// Mitsubishi GX Works2 project: STW_4Counter_Structure_V3   PLC: FX3U/FX3UC

// task Task_01 (event TRUE, interval 0, priority 31): POU_01

PROGRAM POU_01
VAR
  FDCounter_1 : FDCounter;
  FDCounter_2 : FDCounter;
  FDCounter_3 : FDCounter;
  FDCounter_4 : FDCounter;
  FDCounter_5 : FDCounter;
  FDCounter_6 : FDCounter;
  FDCounter_7 : FDCounter;
  FDCounter_8 : FDCounter;
END_VAR
(* structured ladder/FBD written out as ST: instructions are called as NAME(EN, inputs, outputs); _pN, _eN, _tN stand for wires *)
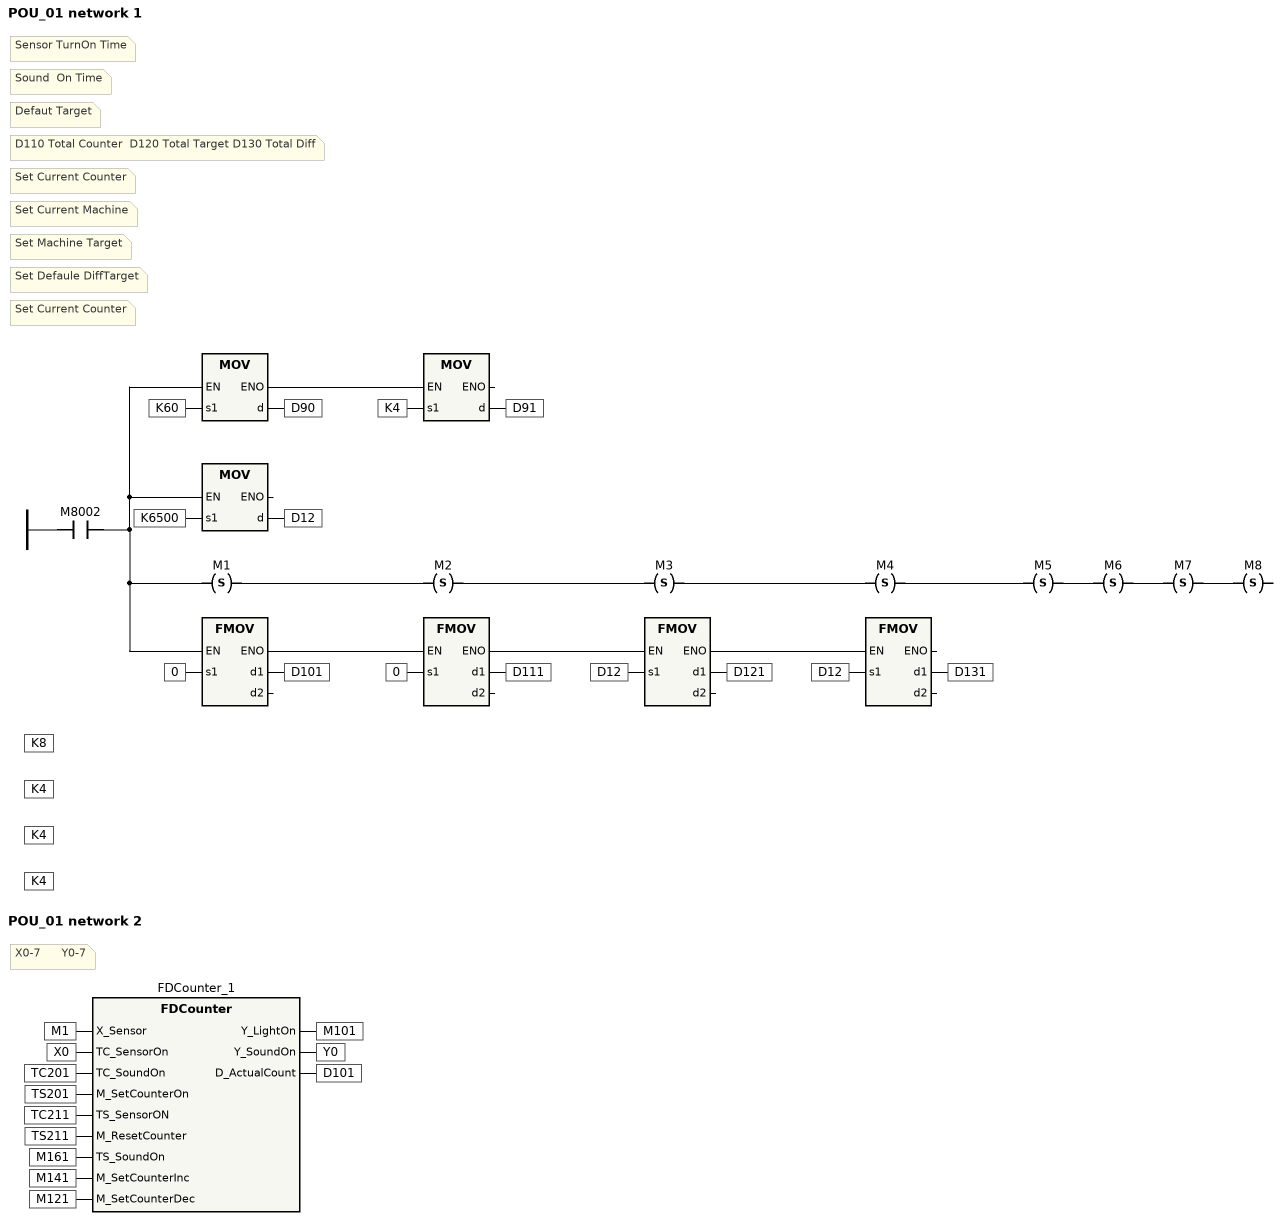
(* network 1 *)
(* Sensor TurnOn Time *)
(* Sound  On Time *)
(* Defaut Target *)
(* D110 Total Counter  D120 Total Target D130 Total Diff *)
(* Set Current Counter *)
(* Set Current Machine *)
(* Set Machine Target *)
(* Set Defaule DiffTarget *)
(* Set Current Counter *)
_e1 := MOV(M8002, K60, D90);
MOV(_e1, K4, D91);
MOV(M8002, K6500, D12);
_e2 := FMOV(M8002, 0, D101, _open);
_e3 := FMOV(_e2, 0, D111, _open);
_e4 := FMOV(_e3, D12, D121, _open);
FMOV(_e4, D12, D131, _open);
SET(M8002, M1);
SET(M8002, M2);
SET(M8002, M3);
SET(M8002, M4);
SET(M8002, M5);
SET(M8002, M6);
SET(M8002, M7);
SET(M8002, M8);
(* not connected to any output: K8, K4, K4, K4 *)
(* network 2 *)
(* X0-7      Y0-7 *)
FDCounter_1(X_Sensor := M1, TC_SensorOn := X0, TC_SoundOn := TC201, M_SetCounterOn := TS201, TS_SensorON := TC211, M_ResetCounter := TS211, TS_SoundOn := M161, M_SetCounterInc := M141, M_SetCounterDec := M121, Y_LightOn => M101, Y_SoundOn => Y0, D_ActualCount => D101);
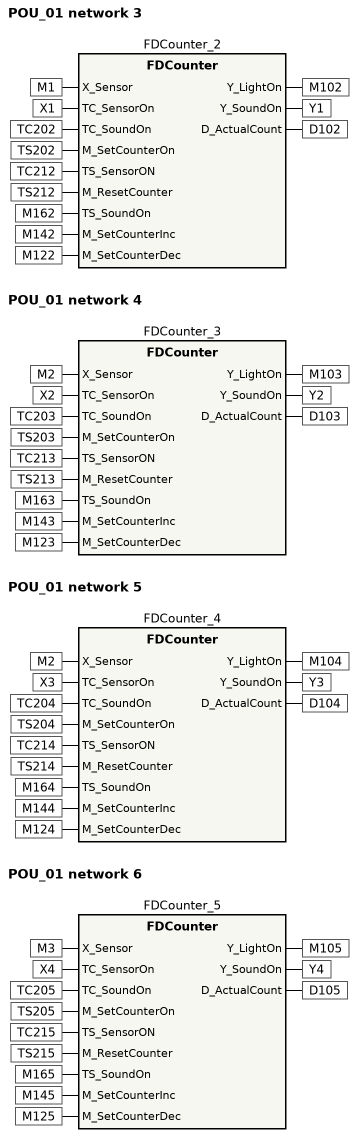
(* network 3 *)
FDCounter_2(X_Sensor := M1, TC_SensorOn := X1, TC_SoundOn := TC202, M_SetCounterOn := TS202, TS_SensorON := TC212, M_ResetCounter := TS212, TS_SoundOn := M162, M_SetCounterInc := M142, M_SetCounterDec := M122, Y_LightOn => M102, Y_SoundOn => Y1, D_ActualCount => D102);
(* network 4 *)
FDCounter_3(X_Sensor := M2, TC_SensorOn := X2, TC_SoundOn := TC203, M_SetCounterOn := TS203, TS_SensorON := TC213, M_ResetCounter := TS213, TS_SoundOn := M163, M_SetCounterInc := M143, M_SetCounterDec := M123, Y_LightOn => M103, Y_SoundOn => Y2, D_ActualCount => D103);
(* network 5 *)
FDCounter_4(X_Sensor := M2, TC_SensorOn := X3, TC_SoundOn := TC204, M_SetCounterOn := TS204, TS_SensorON := TC214, M_ResetCounter := TS214, TS_SoundOn := M164, M_SetCounterInc := M144, M_SetCounterDec := M124, Y_LightOn => M104, Y_SoundOn => Y3, D_ActualCount => D104);
(* network 6 *)
FDCounter_5(X_Sensor := M3, TC_SensorOn := X4, TC_SoundOn := TC205, M_SetCounterOn := TS205, TS_SensorON := TC215, M_ResetCounter := TS215, TS_SoundOn := M165, M_SetCounterInc := M145, M_SetCounterDec := M125, Y_LightOn => M105, Y_SoundOn => Y4, D_ActualCount => D105);
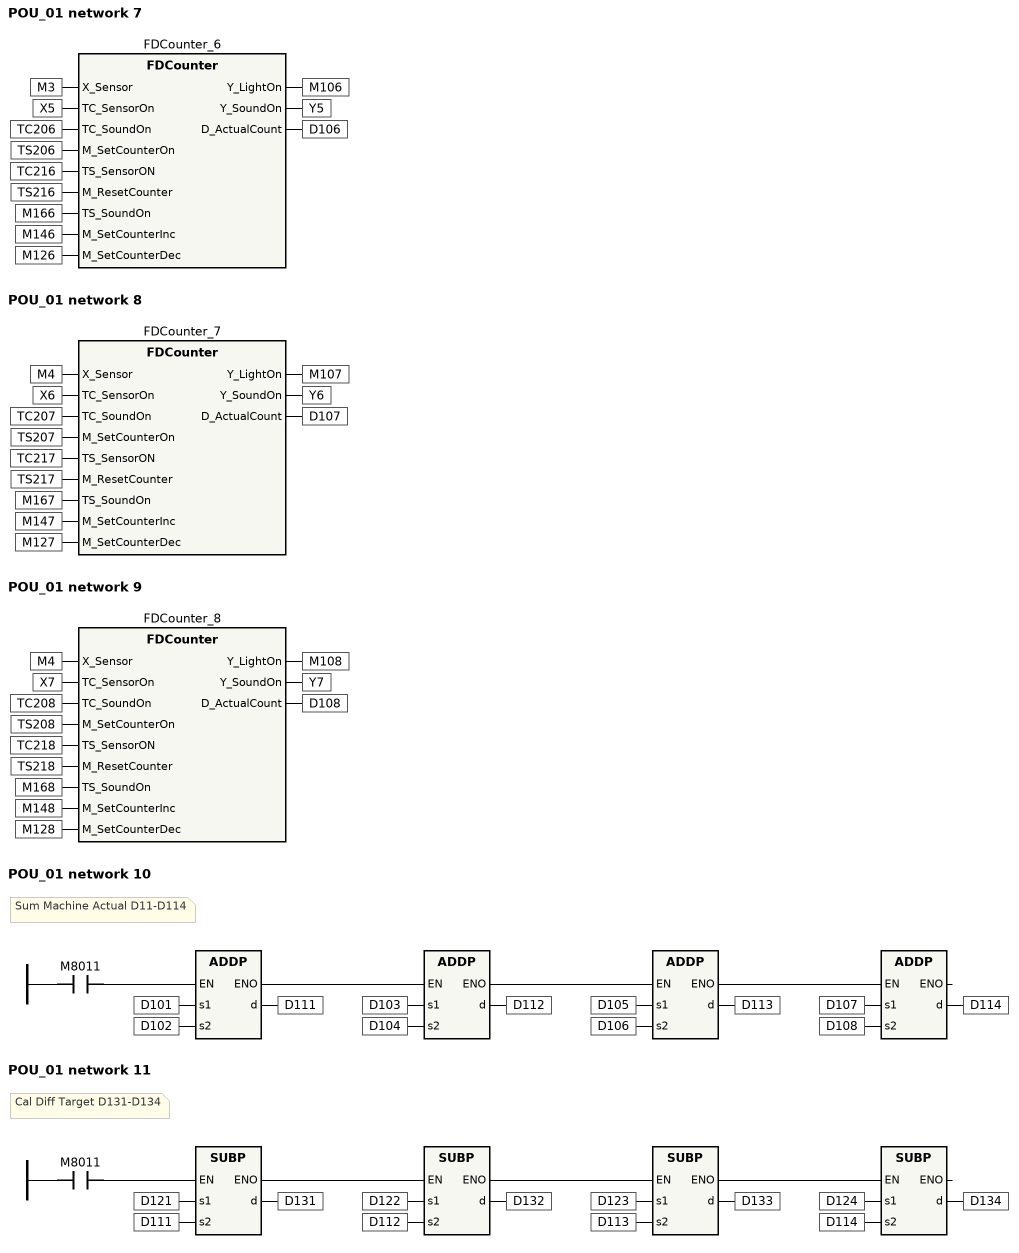
(* network 7 *)
FDCounter_6(X_Sensor := M3, TC_SensorOn := X5, TC_SoundOn := TC206, M_SetCounterOn := TS206, TS_SensorON := TC216, M_ResetCounter := TS216, TS_SoundOn := M166, M_SetCounterInc := M146, M_SetCounterDec := M126, Y_LightOn => M106, Y_SoundOn => Y5, D_ActualCount => D106);
(* network 8 *)
FDCounter_7(X_Sensor := M4, TC_SensorOn := X6, TC_SoundOn := TC207, M_SetCounterOn := TS207, TS_SensorON := TC217, M_ResetCounter := TS217, TS_SoundOn := M167, M_SetCounterInc := M147, M_SetCounterDec := M127, Y_LightOn => M107, Y_SoundOn => Y6, D_ActualCount => D107);
(* network 9 *)
FDCounter_8(X_Sensor := M4, TC_SensorOn := X7, TC_SoundOn := TC208, M_SetCounterOn := TS208, TS_SensorON := TC218, M_ResetCounter := TS218, TS_SoundOn := M168, M_SetCounterInc := M148, M_SetCounterDec := M128, Y_LightOn => M108, Y_SoundOn => Y7, D_ActualCount => D108);
(* network 10 *)
(* Sum Machine Actual D11-D114 *)
_e1 := ADDP(M8011, D101, D102, D111);
_e2 := ADDP(_e1, D103, D104, D112);
_e3 := ADDP(_e2, D105, D106, D113);
ADDP(_e3, D107, D108, D114);
(* network 11 *)
(* Cal Diff Target D131-D134 *)
_e1 := SUBP(M8011, D121, D111, D131);
_e2 := SUBP(_e1, D122, D112, D132);
_e3 := SUBP(_e2, D123, D113, D133);
SUBP(_e3, D124, D114, D134);
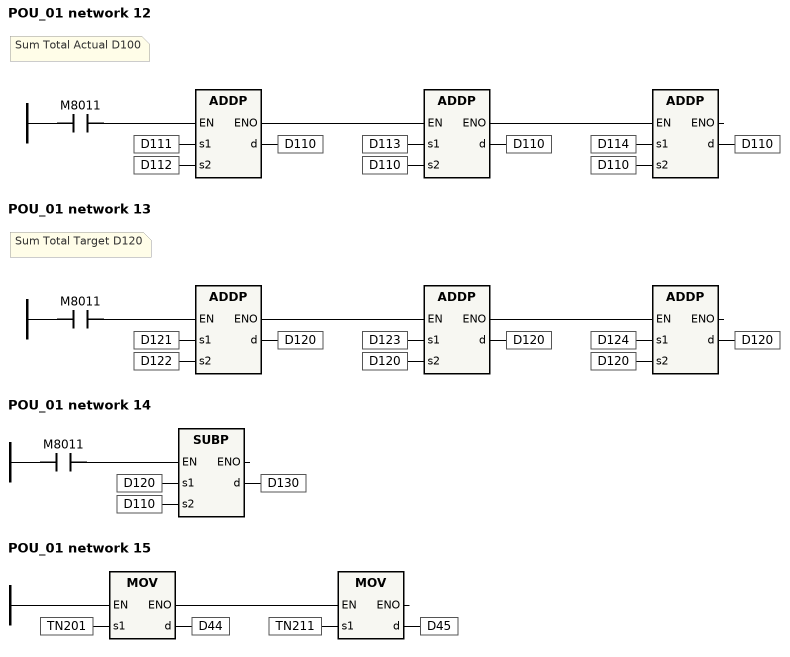
(* network 12 *)
(* Sum Total Actual D100 *)
_e1 := ADDP(M8011, D111, D112, D110);
_e2 := ADDP(_e1, D113, D110, D110);
ADDP(_e2, D114, D110, D110);
(* network 13 *)
(* Sum Total Target D120 *)
_e1 := ADDP(M8011, D121, D122, D120);
_e2 := ADDP(_e1, D123, D120, D120);
ADDP(_e2, D124, D120, D120);
(* network 14 *)
SUBP(M8011, D120, D110, D130);
(* network 15 *)
_e1 := MOV(TRUE, TN201, D44);
MOV(_e1, TN211, D45);
END_PROGRAM

FUNCTION_BLOCK FDCounter
VAR_INPUT
  X_Sensor : BOOL;
END_VAR
VAR_OUTPUT
  Y_LightOn : BOOL;
  Y_SoundOn : BOOL;
END_VAR
VAR_INPUT
  TC_SensorOn : BOOL;
  TC_SoundOn : BOOL;
  M_SetCounterOn : BOOL;
  TS_SensorON : BOOL;
  M_ResetCounter : BOOL;
  TS_SoundOn : BOOL;
  M_SetCounterInc : BOOL;
  M_SetCounterDec : BOOL;
END_VAR
VAR_OUTPUT
  D_ActualCount : INT;
END_VAR
(* structured ladder/FBD written out as ST: instructions are called as NAME(EN, inputs, outputs); _pN, _eN, _tN stand for wires *)
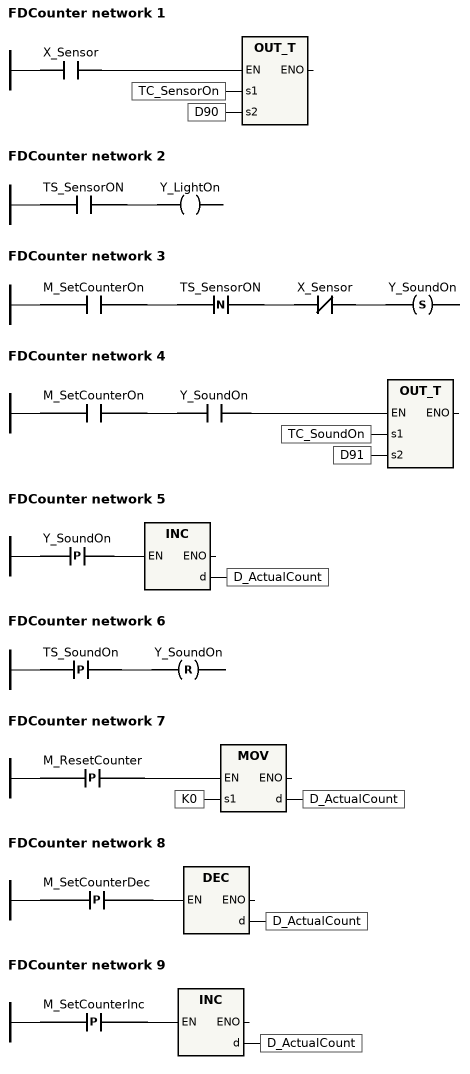
(* network 1 *)
OUT_T(X_Sensor, TC_SensorOn, D90);
(* network 2 *)
Y_LightOn := TS_SensorON;
(* network 3 *)
SET(M_SetCounterOn AND LDF(TRUE, TS_SensorON) AND NOT X_Sensor, Y_SoundOn);
(* network 4 *)
OUT_T(M_SetCounterOn AND Y_SoundOn, TC_SoundOn, D91);
(* network 5 *)
INC(LDP(TRUE, Y_SoundOn), D_ActualCount);
(* network 6 *)
RST(LDP(TRUE, TS_SoundOn), Y_SoundOn);
(* network 7 *)
MOV(LDP(TRUE, M_ResetCounter), K0, D_ActualCount);
(* network 8 *)
DEC(LDP(TRUE, M_SetCounterDec), D_ActualCount);
(* network 9 *)
INC(LDP(TRUE, M_SetCounterInc), D_ActualCount);
END_FUNCTION_BLOCK

// device comments not shown above
D11  ; DK_TC_SensorON
